FUNCTION_BLOCK DELAY_MS (* Simple FB with one algorithm *)
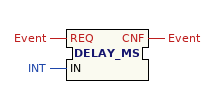
  EVENT_INPUT
    REQ; (* Normal Execution Request *)
  END_EVENT
  EVENT_OUTPUT
    CNF; (* Execution Confirmation *)
  END_EVENT
  VAR_INPUT
    IN : INT; (* Delay Time ms *)
  END_VAR
END_FUNCTION_BLOCK
